FUNCTION_BLOCK FB_Sensor_NO
VAR_INPUT
END_VAR
VAR_OUTPUT
END_VAR
VAR
END_VAR

END_FUNCTION_BLOCK

(* stored: Version 1.1.0.1, ProductVersion 3.1.4024.12
   POU FB_Sensor_NO: Id {4d1a23dc-7a7e-4d31-8b3b-1d870d57f715}, SpecialFunc None *)
